// ==============================================================================
// DB_SimConfig - Конфігурація симуляторів механізмів
// ==============================================================================
// Версія: 2.0.0
// Дата: 2026-01-29
// ==============================================================================
// Призначення:
//   Зберігає налаштування симуляції для всіх типів механізмів
//   RETAIN - налаштування зберігаються після перезавантаження CPU
//
// Розділення відповідальності:
//   - DB_SimMechs (NON_RETAIN) - runtime стан (мотор працює, розгін, аварії)
//   - DB_SimConfig (RETAIN) - налаштування (часи, увімкнення симуляції)
//
// Використання:
//   1. Налаштуйте параметри у DB_SimConfig через HMI або онлайн-редагування
//   2. Викликайте FC_Sim<Type>, передаючи параметри з конфігу
// ==============================================================================

DATA_BLOCK "DB_SimConfig"
{ S7_Optimized_Access := 'TRUE' }
VERSION : 2.0

VAR
    // === Масиви конфігурацій ===

    // Редлери
    Redler : ARRAY[0.."REDLERS_COUNT"] OF "UDT_SimRedlerConfig";

    // Норії
    Noria : ARRAY[0.."NORIAS_COUNT"] OF "UDT_SimNoriaConfig";

    // Вентилятори
    Fan : ARRAY[0.."FANS_COUNT"] OF "UDT_SimFanConfig";

END_VAR

BEGIN
    // === Початкові налаштування (приклади) ===

    // Редлер 0 - увімкнено для тестування
    Redler[0].Enable := TRUE;
    Redler[0].StartupTime_ms := 3000;
    Redler[0].StopTime_ms := 2000;
    Redler[0].SimFault_Breaker := FALSE;
    Redler[0].FaultTime_Breaker_ms := 10000;
    Redler[0].SimFault_Overflow := FALSE;
    Redler[0].FaultTime_Overflow_ms := 15000;


	// Редлер 1 - увімкнено для тестування
    Redler[1].Enable := TRUE;
    Redler[1].StartupTime_ms := 3000;
    Redler[1].StopTime_ms := 2000;
    Redler[1].SimFault_Breaker := FALSE;
    Redler[1].FaultTime_Breaker_ms := 10000;
    Redler[1].SimFault_Overflow := FALSE;
    Redler[1].FaultTime_Overflow_ms := 15000;



    NORIA[0].Enable                 := TRUE;  // увімкнути симуляцію цієї норії
    NORIA[0].StartupTime_ms         := 4000;   // час розгону до робочої швидкості (мс)
    NORIA[0].StopTime_ms            := 3000;   // час вибігу після зупинки (мс)
    NORIA[0].SimFault_Breaker       := FALSE;  // увімкнути симуляцію FLT_BREAKER
    NORIA[0].FaultTime_Breaker_ms   := 10000;  // час до аварії від пуску мотора (мс)
    NORIA[0].SimFault_Alignment     := FALSE;  // увімкнути симуляцію FLT_ALIGNMENT
    NORIA[0].FaultTime_Alignment_ms := 20000; // час до аварії від пуску (мс)
    NORIA[0].ManualReset            := FALSE;  // кнопка скидання латчованих аварій





    // Решта механізмів за замовчуванням вимкнені (Enable := FALSE)

END_DATA_BLOCK
